PROGRAM Environment
VAR_OUTPUT
	WindSpeed,
	WindDirection,
	Temperature,
	Humidity,
	Pressure,
	TemperatureDome,
	HumidityDome,
	DewpointDome:	REAL;
	
	Rain:	BOOL;
	Rain_analog:	REAL;
	WeatherBad:	BOOL;
END_VAR
VAR
	WindEvent,
	HumidityEvent,
	HumidityDomeEvent,
	PrecipitationEvent,
	DewpointEvent: FB_Eventlog;
	WindAverage,
	Wind5sAverage,
	WindDirectionAverage,
	HumidityAverage,
	HumidityDomeAverage,
	PressureAverage,
	Rain_average: FB_TimeAverage;
	RainDelay:	TON;
	sunpos:		FB_SUNPOS;
	eq2hor2:	FB_EQ2HOR2;
	avg_wind, max_wind: REAL;
	MQTTTimer : TON := (PT:=T#5S);
	sPayloadPub: STRING(255) := '';
END_VAR

(* convert raw Sensor values to real values *)
WindSpeed := 		F_YREAL(GVL_Environment.rawWindSpeed, 		0, 32767,   0.0, 50.0); // m/s
WindDirection :=	F_YREAL(GVL_Environment.rawWindDirection, 	0, 32767,   0.0, 360.0); // °
Temperature :=  	F_YREAL(GVL_Environment.rawTemperature, 	0, 32767, -30.0, 70.0); // °C -40...80?
Humidity :=			F_YREAL(GVL_Environment.rawHumidity, 		0, 32767,   0.0, 100.0); // %
Pressure := 		F_YREAL(GVL_Environment.rawPressure,		0, 32767, 600.0, 1520.0); // mBar 

HumidityDome :=		F_YREAL(GVL_Environment.rawHumidityDome, 		0, 32767,   0.0, 100.0); // %
TemperatureDome :=  F_YREAL(GVL_Environment.rawTemperatureDome, 	0, 32767, -30.0, 70.0); // °C

DewpointDome := 	F_Dewpoint(HumidityDome, TemperatureDome);

RainDelay(IN := NOT GVL_Environment.rawRain, PT := T#10S, Q => Rain);

WindAverage(IN := WindSpeed, PT := T#3M, AVG => avg_wind, MAXAVG => max_wind);
Wind5sAverage(IN := WindSpeed, PT := T#5S);
WindDirectionAverage(IN := WindDirection, PT := T#5S);
HumidityAverage(IN := Humidity, PT := T#2M);
// TemperatureAverage(IN := Temperature, PT := T#5M);
PressureAverage(IN := Pressure, PT := T#5S);

HumidityDomeAverage(IN := HumidityDome, PT := T#2M);

Rain_average(IN := BOOL_TO_INT(NOT GVL_Environment.rawRain) * 100.0, PT := T#60s, AVG => Rain_analog);

WeatherBad := Rain OR
				HumidityAverage.AVG >= 80.0 OR
				HumidityDomeAverage.AVG >= 80.0 OR
				WindAverage.AVG*2.0 > 10.0 OR
				max_wind*2 > 15.0;

IF WeatherBad AND DomeControl.DomeOpened THEN
	DomeControl.CloseDome := TRUE;
END_IF

sunpos(JD := TelescopeControl.jd);
eq2hor2(alpha := sunpos.RA,
	delta := sunpos.Dec,
	lon := TelescopeControl.longitude,
	lat := TelescopeControl.latitude,
	JD := TelescopeControl.jd);

MQTTTimer(IN:=TRUE);
IF MQTTTimer.Q THEN // publish new payload every second
	MQTTTimer(IN:=FALSE);
	sPayloadPub := 'environment,location=roof,host=CX-4E6032 ';
	sPayloadPub := APPEND(sPayloadPub, 'OutsideTemperature=', LREAL_TO_FMTSTR(Temperature, 2, TRUE));
	sPayloadPub := APPEND(sPayloadPub, ',OutsideHumidity=', LREAL_TO_FMTSTR(Humidity, 1, TRUE));
	sPayloadPub := APPEND(sPayloadPub, ',WindSpeed=', LREAL_TO_FMTSTR(Wind5sAverage.AVG, 1, TRUE));
	sPayloadPub := APPEND(sPayloadPub, ',WindSpeedMax=', LREAL_TO_FMTSTR(Wind5sAverage.MAXAVG, 1, TRUE));
	sPayloadPub := APPEND(sPayloadPub, ',WindDirection=', LREAL_TO_FMTSTR(WindDirectionAverage.AVG, 1, TRUE));
	sPayloadPub := APPEND(sPayloadPub, ',Pressure=', LREAL_TO_FMTSTR(PressureAverage.AVG, 2, TRUE));
	sPayloadPub := APPEND(sPayloadPub, ',Rain=', BOOL_TO_STRING(Rain));
	sPayloadPub := APPEND(sPayloadPub, ',RainAnalog=', LREAL_TO_FMTSTR(Rain_analog, 1, TRUE));
	
	MQTTCommunication.fbMqttClient.Publish(	
					sTopic:= 'RoboTel/Telemetry', 
					pPayload:= ADR(sPayloadPub), 
					nPayloadSize:= LEN2(ADR(sPayloadPub)),
					eQoS:= TcIotMqttQos.AtMostOnceDelivery,
					bRetain:= FALSE, 
					bQueue:= FALSE );
					
	sPayloadPub := 'dome,location=dome,host=CX-4E6032 ';
	sPayloadPub := APPEND(sPayloadPub, 'DomeTemperature=', LREAL_TO_FMTSTR(TemperatureDome, 2, TRUE));
	sPayloadPub := APPEND(sPayloadPub, ',DomeHumidity=', LREAL_TO_FMTSTR(HumidityDome, 1, TRUE));
	sPayloadPub := APPEND(sPayloadPub, ',WeatherBad=', BOOL_TO_STRING(WeatherBad));
	
	MQTTCommunication.fbMqttClient.Publish(	
					sTopic:= 'RoboTel/Telemetry', 
					pPayload:= ADR(sPayloadPub), 
					nPayloadSize:= LEN2(ADR(sPayloadPub)),
					eQoS:= TcIotMqttQos.AtMostOnceDelivery,
					bRetain:= FALSE, 
					bQueue:= FALSE );

END_IF

WindEvent(	Trigger := avg_wind > 10.0, 
			Level := ADSLOG_MSGTYPE_WARN,
			FormatString := 'Wind Speed: %s',
			OnMessage := LREAL_TO_FMTSTR(WindSpeed, 2, TRUE),
			OffMessage := 'OK',
			OffLevel := ADSLOG_MSGTYPE_HINT);

HumidityEvent(	Trigger :=  HumidityAverage.AVG>= 80.0, 
				Level := ADSLOG_MSGTYPE_WARN,
				FormatString := 'Humidity: %s',
				OnMessage := LREAL_TO_FMTSTR( HumidityAverage.AVG, 1, TRUE),
				OffMessage := 'OK',
				OffLevel := ADSLOG_MSGTYPE_HINT);

// azimuth encoder starts to fail at 65% humidity
HumidityDomeEvent(	Trigger :=  HumidityDomeAverage.AVG>= 65.0, 
				Level := ADSLOG_MSGTYPE_WARN,
				FormatString := 'Humidity in Dome: %s',
				OnMessage := LREAL_TO_FMTSTR( HumidityDomeAverage.AVG, 1, TRUE),
				OffMessage := 'OK',
				OffLevel := ADSLOG_MSGTYPE_HINT);

				
PrecipitationEvent(	Trigger := WeatherBad, 
					Level := ADSLOG_MSGTYPE_WARN,
					FormatString := 'The weather is %s',
					OnMessage := 'BAD.',
					OffMessage := 'OK.');

DewPointEvent( Trigger := TemperatureDome < DewpointDome,
				Level := ADSLOG_MSGTYPE_WARN,
				FormatString := 'Dewpoint in Dome below ambient Temperature: %s',
				OnMessage := LREAL_TO_FMTSTR( DewpointDome, 1, TRUE),
				OffMessage := 'OK',
				OffLevel := ADSLOG_MSGTYPE_HINT);

END_PROGRAM

(* stored: Version 1.1.0.1, ProductVersion 3.1.4024.9
   POU Environment: Id {03869fa8-1755-402e-a7ee-189c483e0438}, SpecialFunc None *)
